FUNCTION_BLOCK SimpleBatteryModel (* Simple battery model for pre-simulation of charge/discharge. *)
  (* Standard: 61499-2; Description: Simple battery model for pre-simulation of charge/discharge. Simulates a charge/discharge requests with an array PV surplus/deficits, a given feed-in and/or load limitation and the battery's current state of charge. The simulation occurs based on characteristics, such as battery efficiency, inverter efficiency, etc. NOTE: It is recommended to replace this model with the manufacturer's battery model for more precise results. IEC 61499 implementation of the "PVprog" algorithm. Original version's MIT license: Copyright (c) 2016 Joseph Bergner, Johannes Weniger, Tjarko Tjaden Permission is hereby granted, free of charge, to any person obtaining a copy of this software and associated documentation files (the "Software"), to deal in the Software without restriction, including without limitation the rights to use, copy, modify, merge, publish, distribute, sublicense, and/or sell copies of the Software, and to permit persons to whom the Software is furnished to do so, subject to the following conditions: The above copyright notice and this permission notice shall be included in all copies or substantial portions of the Software. THE SOFTWARE IS PROVIDED "AS IS", WITHOUT WARRANTY OF ANY KIND, EXPRESS OR IMPLIED, INCLUDING BUT NOT LIMITED TO THE WARRANTIES OF MERCHANTABILITY, FITNESS FOR A PARTICULAR PURPOSE AND NONINFRINGEMENT. IN NO EVENT SHALL THE AUTHORS OR COPYRIGHT HOLDERS BE LIABLE FOR ANY CLAIM, DAMAGES OR OTHER LIABILITY, WHETHER IN AN ACTION OF CONTRACT, TORT OR OTHERWISE, ARISING FROM, OUT OF OR IN CONNECTION WITH THE SOFTWARE OR THE USE OR OTHER DEALINGS IN THE SOFTWARE. *)
  (* Version 1.0, 2017-05-17, Marc Jakobi, HTW Berlin *)
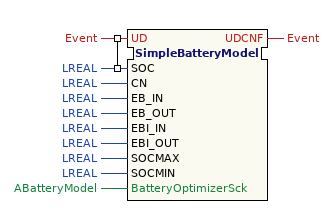
  EVENT_INPUT
    UD WITH SOC; (* Update Request *)
  END_EVENT
  EVENT_OUTPUT
    UDCNF; (* Update Confirmation *)
  END_EVENT
  VAR_INPUT
    SOC : LREAL := 0.2; (* State of charge of the battery [0..1] *)
    CN : LREAL; (* Nominal battery capacity (energy) in kWh *)
    EB_IN : LREAL := 0.96; (* Battery efficiency when charging [0..1] *)
    EB_OUT : LREAL := 0.96; (* Battery efficiency when discharging [0..1] *)
    EBI_IN : LREAL := 0.96; (* Battery inverter efficiency when charging [0..1] *)
    EBI_OUT : LREAL := 0.96; (* Battery inverter efficiency when discharging [0..1] *)
    SOCMAX : LREAL := 1; (* Upper limit to SOC (as specified by manufacturer) [0..1] *)
    SOCMIN : LREAL := 0.2; (* Lower limit to SOC (as specified by manufacturer) [0..1] *)
  END_VAR
  SOCKETS
    BatteryOptimizerSck : ABatteryModel; (* Link to BatteryOptimizer *)
  END_SOCKETS
  VAR
    CIN : LREAL; (* Energy stored in battery before simulation in kWh *)
    CMAX : LREAL; (* Maximum capacity in kWh *)
    CMIN : LREAL; (* Minimum capacity in kWh *)
  END_VAR
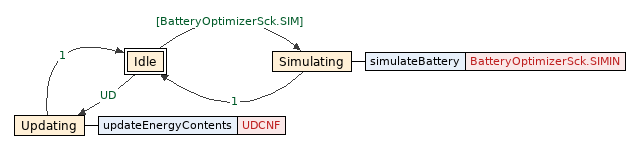
  EC_STATES
    Idle; (* Initial State *)
    Simulating : simulateBattery -> BatteryOptimizerSck.SIMIN; (* Normal execution *)
    Updating : updateEnergyContents -> UDCNF;
  END_STATES
  EC_TRANSITIONS
    Idle TO Simulating := [BatteryOptimizerSck.SIM];
    Simulating TO Idle := 1;
    Updating TO Idle := 1;
    Idle TO Updating := UD;
  END_TRANSITIONS
  ALGORITHM simulateBattery IN ST: (* Simulates battery charging/discharging *)
IF BatteryOptimizerSck.ECD > 0 THEN
	BatteryOptimizerSck.CSIM := CIN + EB_IN * EBI_IN * BatteryOptimizerSck.ECD; // charge
	IF BatteryOptimizerSck.CSIM > CMAX THEN
		BatteryOptimizerSck.CSIM := CMAX; // limit to max capacity
	END_IF;
ELSIF BatteryOptimizerSck.ECD < 0 THEN
	BatteryOptimizerSck.CSIM := CIN + EB_OUT * EBI_OUT * BatteryOptimizerSck.ECD; // discharge
	IF BatteryOptimizerSck.CSIM < CMIN THEN
		BatteryOptimizerSck.CSIM := CMIN; // limit to min capacity
	END_IF;
ELSE
	BatteryOptimizerSck.CSIM := CIN;
END_IF;
  END_ALGORITHM
  ALGORITHM updateEnergyContents IN ST: (* Updates the battery's energy contents upon arrival of a new SOC measurement *)
CIN := SOC * CN;
CMAX := SOCMAX * CN;
CMIN := SOCMIN * CN;
  END_ALGORITHM
END_FUNCTION_BLOCK
